INTERFACE ISequence
// Copyright (c) 2024 Loupe (https://loupe.team), provided under the MIT License.

{attribute 'monitoring' := 'call'}
PROPERTY CurrentStep : ENUM
GET
END_GET
END_PROPERTY

METHOD DoStep : ENUM
VAR
END_VAR
END_METHOD

METHOD OnAbort : BOOL
VAR_INPUT
    nextStep : ENUM;
END_VAR
END_METHOD

METHOD OnEntry : BOOL
VAR_INPUT
END_VAR
END_METHOD

METHOD OnError : BOOL
VAR_INPUT
    nextStep : ENUM;
END_VAR
END_METHOD

METHOD OnExit : BOOL
VAR_INPUT
END_VAR
END_METHOD

METHOD OnFailure : BOOL
VAR_INPUT
    nextStep : ENUM;
END_VAR
END_METHOD

METHOD OnSuccess : BOOL
VAR_INPUT
    nextStep : ENUM;
END_VAR
END_METHOD

METHOD RequestStep : BOOL
VAR_INPUT
    nextStep : ENUM;
END_VAR
END_METHOD

METHOD RequestStepClear : BOOL
VAR_INPUT
    nextStep : ENUM;
END_VAR
END_METHOD

METHOD SequenceAbort : BOOL
VAR_INPUT
    ErrorCode : DINT;
    ErrorMessage : STRING;
END_VAR
END_METHOD

METHOD SequenceComplete : BOOL
VAR_INPUT
END_VAR
END_METHOD

METHOD SequenceError : BOOL
VAR_INPUT
    ErrorCode : INT;
    ErrorMessage : STRING;
END_VAR
END_METHOD

METHOD StartSequence : BOOL
VAR_INPUT
	Status : IPLCopenCaller;
END_VAR
END_METHOD

END_INTERFACE

(* stored: Version 1.1.0.1
   Itf ISequence: Id {ec403192-db1e-410a-9f94-aa5afd69329b}
   Folder Callbacks: Id {3d1e23ba-0316-470f-8744-3aa607d72bad}
   Folder StateControl: Id {daaf35c2-6411-4d82-aef2-a15497701697}
   Property CurrentStep: Id {d83302e6-d8e8-46af-86eb-9a1fd884af7b}
   Get Get: Id {ab2da43a-d96f-44aa-8e36-8c2ba2c37047}
   Method DoStep: Id {9a34277b-a3ad-4319-a578-90c522c3c623}
   Method OnAbort: Id {4445ff1a-fbfc-4467-ae59-52d6282d62cc}
   Method OnEntry: Id {151235a9-806e-47c6-9584-1ba6690c0af0}
   Method OnError: Id {bcf3cc66-e294-4626-a88a-229a42065635}
   Method OnExit: Id {7a1ed197-67b1-4a9f-b7b9-e80cf5833314}
   Method OnFailure: Id {0fd686e6-f999-4918-9b3d-8a51abb3cd5a}
   Method OnSuccess: Id {82c8d03a-450e-4fab-9845-0d89e2f94a52}
   Method RequestStep: Id {eda50567-af34-458e-89ce-ac3a3abf3610}
   Method RequestStepClear: Id {e59012ec-24ed-47da-8aaf-87ba4a553cbc}
   Method SequenceAbort: Id {53bba82b-ae56-4f65-8efe-cc2958f21910}
   Method SequenceComplete: Id {f99ee7a2-4375-4d65-878a-d803b3f40315}
   Method SequenceError: Id {efd40ff7-83f9-47af-a16c-c4732fe53c27}
   Method StartSequence: Id {1cd7451d-fc48-48da-b2a6-3f2d996e06ee} *)
